Yaskawa INFORM job: GET-SHIFT-VALUE-S2-B.JBI

/JOB
//NAME GET-SHIFT-VALUE-S2-B
//POS
///NPOS 0,0,0,1,0,0
///USER 10
///TOOL 0
///POSTYPE USER
///RECTAN
///RCONF 0,0,0,0,0,0,0,0,0,0,0,0,0,0,0,0,0,0,0,0,0,0,0,0
P00049=2.600,0.000,0.000,0.0000,0.0000,0.0000
//INST
///DATE 2018/10/02 07:30
///ATTR SC,RW
///LVARS 0,0,5,0,0,0,0,0
NOP
'***** get shift value
SUB P049 P049
MACRO1 MJ#(1) ARGF103 ARGF30
SET LD000 D030
MUL LD000 100
SETE P049 (1) LD000
END
